// This function has been automatically generated from the project information.
{attribute 'signature_flag' := '1073741824'}
{attribute 'TcGenerated'}
FUNCTION F_GetCompany : WSTRING
VAR_INPUT
	
END_VAR

F_GetCompany := "Poh";

END_FUNCTION

(* stored: Version 1.1.0.1, ProductVersion 3.1.4019.2
   POU F_GetCompany: Id {7583c190-b1d2-4a79-8812-a31ff4496a76}, SpecialFunc None *)
